// TIA Portal V17 export
// export: Created 2026-05-13T16:54:41.6264603Z, ExportSetting WithDefaults, DisplayName Totally Integrated Automation Portal, DisplayVersion V17 Update 4, DisplayName TIA Portal Openness, DisplayVersion V17 Update 4, DisplayName TIA Portal Version Control Interface, DisplayVersion V17, DisplayName SINAMICS Startdrive Advanced, DisplayVersion V17, DisplayName SINAMICS Startdrive G130, G150, S120, S150, SINAMICS MV, S210, DisplayVersion V17, DisplayName SINAMICS Startdrive G110M, G120, G120C, G120D, G120P, G115D, DisplayVersion V17, DisplayName STEP 7 Professional, DisplayVersion V17 Update 4, DisplayName STEP 7 Safety, DisplayVersion V17, DisplayName WinCC Professional, DisplayVersion V17 Update 4
TagTable "PV"
  PV_JF进风温度 : Real  (PLC tag PV.JF进风温度, HMI_连接_1, 1 s)
  PV_JF进风温度写读 : Real  (PLC tag PV.JF进风温度写读, HMI_连接_1, 1 s)
  PV_CF出风温度 : Real  (PLC tag PV.CF出风温度, HMI_连接_1, 1 s)
  PV_WQ尾气温度 : Real  (PLC tag PV.WQ尾气温度, HMI_连接_1, 1 s)
  PV_JF进风温度P : Real  (PLC tag PV.JF进风温度P, HMI_连接_1, 1 s)
  PV_JF进风温度I : Real  (PLC tag PV.JF进风温度I, HMI_连接_1, 1 s)
  PV_JF进风温度D : Real  (PLC tag PV.JF进风温度D, HMI_连接_1, 1 s)
  PV_JL进料泵 : Real  (PLC tag PV.JL进料泵, HMI_连接_1, 1 s)
  PV_JL进料压力 : Real  (PLC tag PV.JL进料压力, HMI_连接_1, 1 s)
  PV_JL进料流量 : Real  (PLC tag PV.JL进料流量, HMI_连接_1, 1 s)
  PV_JF进风压差变送器 : Real  (PLC tag PV.JF进风压差变送器, HMI_连接_1, 1 s)
  PV_BD布袋压差变送器 : Real  (PLC tag PV.BD布袋压差变送器, HMI_连接_1, 1 s)
  PV_ZT主塔压力 : Real  (PLC tag PV.ZT主塔压力, HMI_连接_1, 1 s)
  PV_YF引风反馈 : Real  (PLC tag PV.YF引风反馈, HMI_连接_1, 1 s)
  PV_LX离心雾化 : Real  (PLC tag PV.LX离心雾化, HMI_连接_1, 1 s)
  PV_JL进料速度 : Real  (PLC tag PV.JL进料速度, HMI_连接_1, 1 s)
  PV_YS映射阀开度 : Real  (PLC tag PV.YS映射阀开度, HMI_连接_1, 1 s)
  PV_GX高效压差 : Real  (PLC tag PV.GX高效压差, HMI_连接_1, 1 s)
  PV_BD布袋压差 : Real  (PLC tag PV.BD布袋压差, HMI_连接_1, 1 s)
  PV_ZG总功率 : Real  (PLC tag PV.ZG总功率, HMI_连接_1, 1 s)
  PV_DJ电加热开度 : Real  (PLC tag PV.DJ电加热开度, HMI_连接_1, 1 s)
  PV_RS热水炉温度P : Real  (PLC tag PV.RS热水炉温度P, HMI_连接_1, 1 s)
  PV_RS热水炉温度I : Real  (PLC tag PV.RS热水炉温度I, HMI_连接_1, 1 s)
  PV_RS热水炉温度D : Real  (PLC tag PV.RS热水炉温度D, HMI_连接_1, 1 s)
  PV_RS热水炉开度 : Real  (PLC tag PV.RS热水炉开度, HMI_连接_1, 1 s)
  PV_RS热水炉温度 : Real  (PLC tag PV.RS热水炉温度, HMI_连接_1, 1 s)
  PV_RS热水炉温度写读 : Real  (PLC tag PV.RS热水炉温度写读, HMI_连接_1, 1 s)
  PV_RS热水炉回收温度 : Real  (PLC tag PV.RS热水炉回收温度, HMI_连接_1, 1 s)
  PV_HW恒温系统温度 : Real  (PLC tag PV.HW恒温系统温度, HMI_连接_1, 1 s)
